FUNCTION_BLOCK CNV_SENSOR (* Basic Function Block Type *)
  (* Standard: 61499-2 *)
  (* Version 0.3, 2009-09-15, JHC, Holobloc Inc, Changed transition priorities. *)
  (* Version 0.2, 2003-12-04, JHC, Rockwell Automation, Renamed for better indexing. *)
  (* Version 0.1, 2002-11-05, JHC, Rockwell Automation, Corrected missing ST element in Algorithm REQ. *)
  (* Version 0.0, 2000-05-30, JHC, Rockwell Automation *)
  (* Compiler header: package fb.rt.student; *)
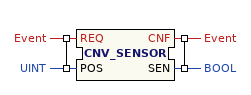
  EVENT_INPUT
    REQ WITH POS; (* Normal Execution Request *)
  END_EVENT
  EVENT_OUTPUT
    CNF WITH SEN; (* Execution Confirmation *)
  END_EVENT
  VAR_INPUT
    POS : UINT; (* Input event qualifier *)
  END_VAR
  VAR_OUTPUT
    SEN : BOOL; (* Output event qualifier *)
  END_VAR
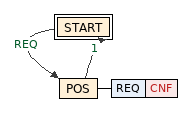
  EC_STATES
    START; (* Initial State *)
    POS : REQ -> CNF;
  END_STATES
  EC_TRANSITIONS
    START TO POS := REQ;
    POS TO START := 1;
  END_TRANSITIONS
  ALGORITHM REQ IN ST: (* Normally executed algorithm *)
IF (POS >= 70) AND (POS < 90) THEN
	SEN := TRUE;
ELSE
	SEN := FALSE;
END_IF;
  END_ALGORITHM
END_FUNCTION_BLOCK
